// TIA Portal V17 export
// export: Created 2024-09-03T21:54:56.0698583Z, ExportSetting WithDefaults, DisplayName Totally Integrated Automation Portal, DisplayVersion V17 Update 7, DisplayName TIA Portal Openness, DisplayVersion V17 Update 7, DisplayName TIA Portal Version Control Interface, DisplayVersion V17, DisplayName SINAMICS Startdrive Advanced, DisplayVersion V17 SP2, DisplayName SINAMICS Startdrive G110M, G120, G120C, G120D, G120P, G115D, DisplayVersion V17 SP2, DisplayName SINAMICS Startdrive G130, G150, S120, S150, SINAMICS MV, S210, DisplayVersion V17 SP2, DisplayName STEP 7 Professional, DisplayVersion V17 Update 7, DisplayName STEP 7 Safety, DisplayVersion V17 Update 6, DisplayName WinCC Advanced / Unified PC, DisplayVersion V17 Update 7
FUNCTION_BLOCK "CycleTimeMeas"   // FB46, FBD
{ S7_Optimized_Access := 'FALSE' }
VERSION : 0.1
// stored: AutoNumber false, IsIECCheckEnabled false, SetENOAutomatically false, UDAEnableTagReadback false
   VAR_INPUT
      StartCycle : Bool;
      ResetHistory : Bool;
   END_VAR
   VAR DB_SPECIFIC
      ActualTime : Time;
      LastTime : Time;
      edge2 : Bool;
      edge1 : Bool;
      Suma : DInt;
      Count : DInt;
      Max : Time;
      Min : Time;
      Average : Time;
      IEC_Timer_0_Instance { S7_SetPoint := 'True'} : TON_TIME;
      History : Array[1..20] of Time;
      NewTime : Bool;
   END_VAR
   VAR_TEMP
      d : DInt;
      i : Int;
   END_VAR
   VAR_TEMP   // added for the SCL form of the ladder/FBD networks
      _w1 : Bool;
   END_VAR
BEGIN

NETWORK
TITLE = Convert time to dint
      L     #ActualTime;
      T     #d;


REGION Network 2: Save cycle time
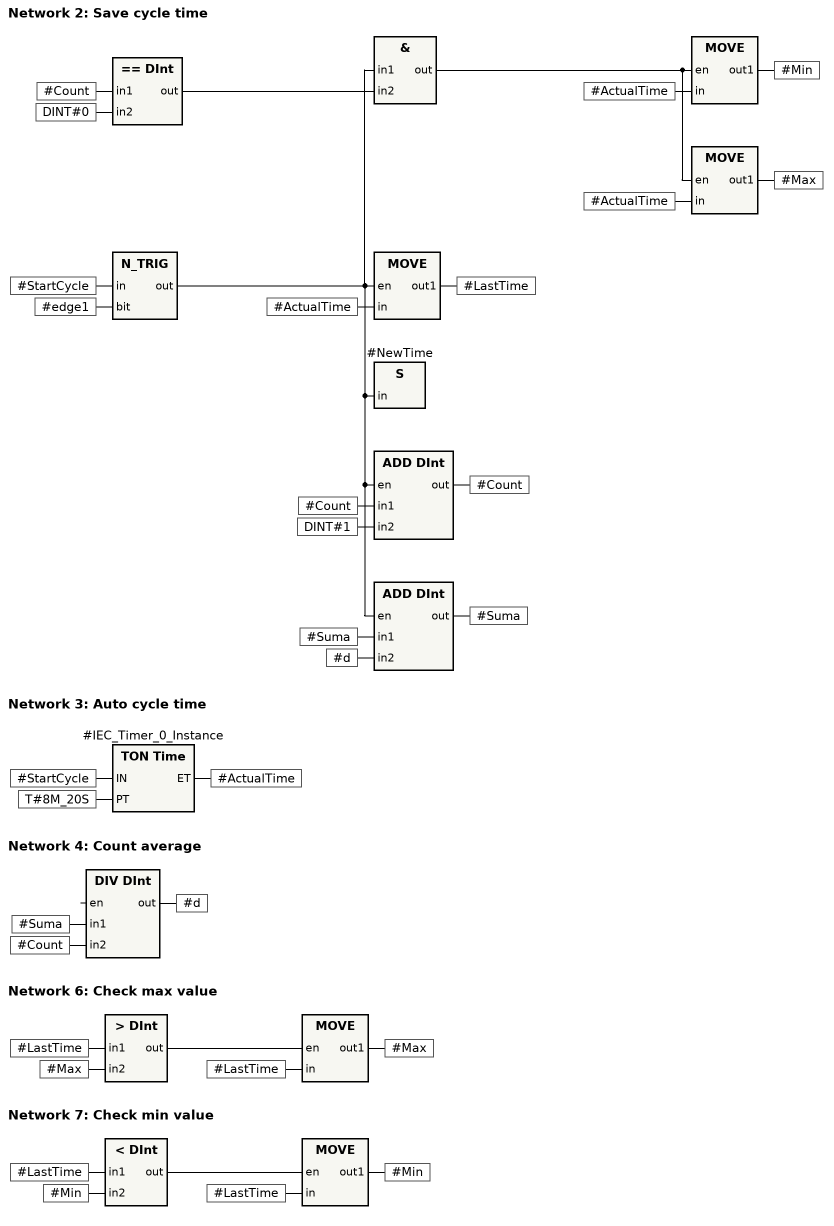
   #_w1 := NOT #StartCycle AND #edge1;   // falling edge
   #edge1 := #StartCycle;
   IF #_w1 THEN
       #LastTime := #ActualTime;
       #NewTime := TRUE;
   END_IF;
   IF #_w1 AND (#Count = DINT#0) THEN
       #Min := #ActualTime;
       #Max := #ActualTime;
   END_IF;
   IF #_w1 THEN
       #Count := #Count + DINT#1;
       #Suma := #Suma + #d;
   END_IF;
END_REGION

REGION Network 3: Auto cycle time
   #IEC_Timer_0_Instance(IN := #StartCycle, PT := T#8M_20S, ET => #ActualTime);   // TON
END_REGION

REGION Network 4: Count average
   #d := #Suma / #Count;
END_REGION

NETWORK
TITLE = Convert dint to time
      L     #d;
      T     #Average;


REGION Network 6: Check max value
   IF #LastTime > #Max THEN #Max := #LastTime; END_IF;
END_REGION

REGION Network 7: Check min value
   IF #LastTime < #Min THEN #Min := #LastTime; END_IF;
END_REGION

REGION Network 8: Reset history
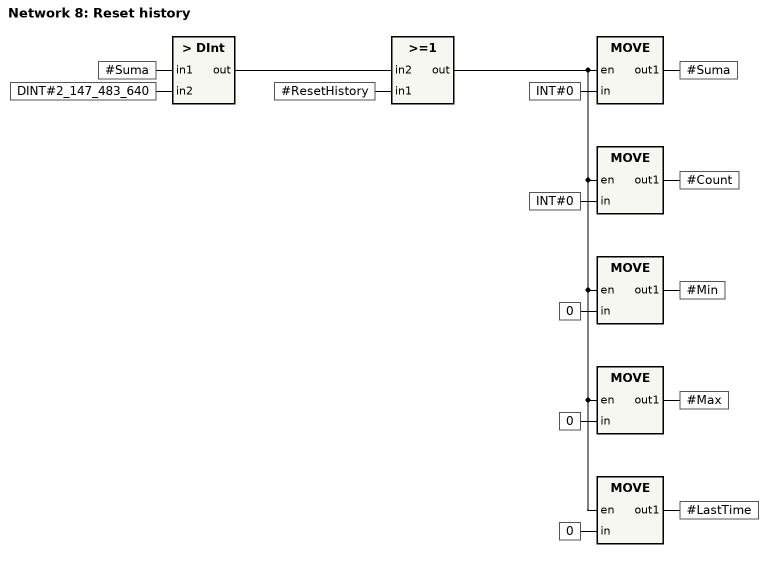
   #_w1 := (#Suma > DINT#2_147_483_640) OR #ResetHistory;
   IF #_w1 THEN
       #Suma := INT#0;
       #Count := INT#0;
       #Min := 0;
       #Max := 0;
       #LastTime := 0;
   END_IF;
END_REGION

REGION Network 10 (SCL)
   IF #NewTime THEN
       FOR #i := 1 TO 19 DO
           #History[21 - #i] := #History[20 - #i];
       END_FOR;
       #History[1] := #LastTime;
   END_IF;
   #NewTime := false;
END_REGION
END_FUNCTION_BLOCK
